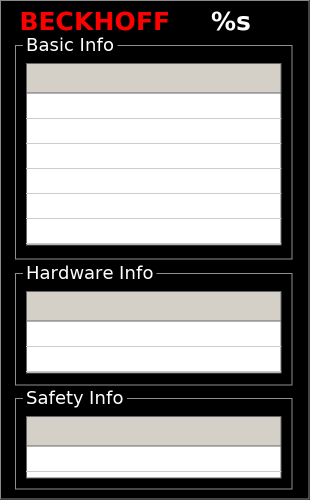
VISUALIZATION PH_SafeDiag_Diagnostic_black  // 310x500
VAR_IN_OUT
	stVisu						: ST_SafeDiag_VisualisationInfos;		
	stSafeDiag					: ST_EL6910_SafeDiag;
END_VAR
    Textfield (10,1 170x40), "BECKHOFF"
    Textfield (171,1 120x40), "%s", text variable: stVisu.sModelNumber
    GroupBox (15,37 277x222), "Basic Info"
        Table (11,26 255x182), data array: stVisu.arrBasicInfos
            p3854506369: stVisu.arrBasicInfos[1,INDEX]
            p1892666644: stVisu.arrBasicInfos[2,INDEX]
    GroupBox (15,265 277x120), "Hardware Info"
        Table (11,26 255x82), data array: stVisu.arrHardwareInfos
            p3854506369: stVisu.arrHardwareInfos[1,INDEX]
            p1892666644: stVisu.arrHardwareInfos[2,INDEX]
    GroupBox (15,390 277x99), "Safety Info"
        Table (11,26 255x62), data array: stVisu.arrSafetyInfos
            p3854506369: stVisu.arrSafetyInfos[1,INDEX]
            p1892666644: stVisu.arrSafetyInfos[2,INDEX]
END_VISUALIZATION

(* stored: Version 1.1.0.1, ProductVersion 3.1.4024.12
   Visu PH_SafeDiag_Diagnostic_black: Id {fa1dfb1d-2f9d-4f14-8325-65e982977165} *)
